{attribute 'qualified_only'}
VAR_GLOBAL
	// Inside cleaner valve
	inValve AT %Q*: BOOL;
	// Outside cleaner valve
	outValve AT %Q*: BOOL;
	
	// ADD COVER SERVO TO SOLUTION
END_VAR

(* stored: Version 1.1.0.1, ProductVersion 3.1.4024.5
   GVL CLEANout: Id {e3f58c5f-7e5d-4c1e-aac9-8e2dda3fc696} *)
